TEXTLIST KPlaceMode
  0 = 'Suction'
  1 = 'Position'
   = ''
END_TEXTLIST

(* stored: Version 1.1.0.1, ProductVersion 3.1.4024.11
   TextList KPlaceMode: Id {8e48e9bf-90a7-4d6c-a5a2-06d0c6db42fd} *)
